// Mitsubishi GX Works2 project: Prog1 IHM_elipse_clp   PLC: FX3U/FX3UC
// Configuração Modbus RTU

PROGRAM MAIN
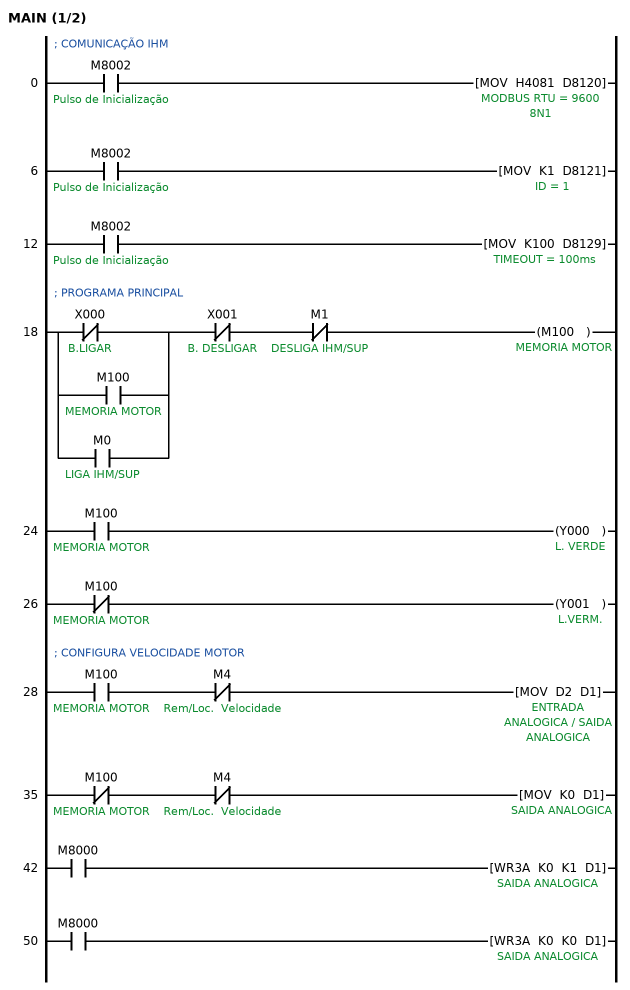
; COMUNICAÇÃO IHM
0     LD      M8002  ; Pulso de Inicialização
      MOV     H4081 D8120  ; MODBUS RTU = 9600 8N1
6     LD      M8002  ; Pulso de Inicialização
      MOV     K1 D8121  ; ID = 1
12    LD      M8002  ; Pulso de Inicialização
      MOV     K100 D8129  ; TIMEOUT = 100ms
; PROGRAMA PRINCIPAL
18    LDI     X000  ; B.LIGAR
      OR      M100  ; MEMORIA MOTOR
      OR      M0  ; LIGA IHM/SUP
      ANI     X001  ; B. DESLIGAR
      ANI     M1  ; DESLIGA IHM/SUP
      OUT     M100  ; MEMORIA MOTOR
24    LD      M100  ; MEMORIA MOTOR
      OUT     Y000  ; L. VERDE
26    LDI     M100  ; MEMORIA MOTOR
      OUT     Y001  ; L.VERM.
; CONFIGURA VELOCIDADE MOTOR
28    LD      M100  ; MEMORIA MOTOR
      ANI     M4  ; Rem/Loc.  Velocidade
      MOV     D2 D1  ; ENTRADA ANALOGICA / SAIDA ANALOGICA
35    LDI     M100  ; MEMORIA MOTOR
      ANI     M4  ; Rem/Loc.  Velocidade
      MOV     K0 D1
42    LD      M8000
      WR3A    K0 K1 D1
50    LD      M8000
      WR3A    K0 K0 D1
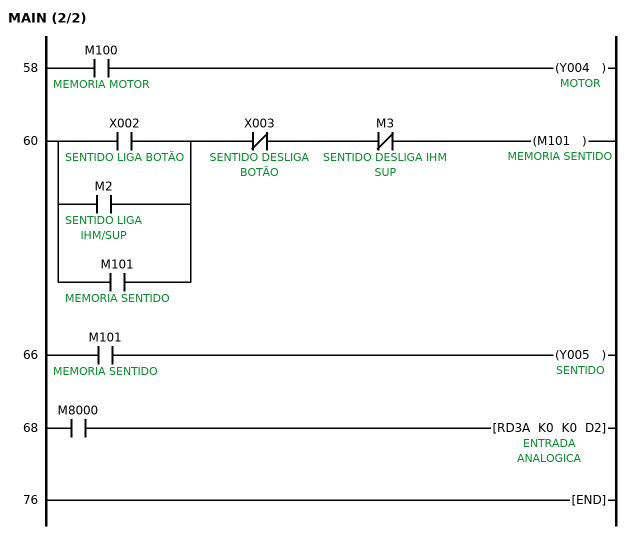
58    LD      M100  ; MEMORIA MOTOR
      OUT     Y004  ; MOTOR
60    LD      X002  ; SENTIDO LIGA BOTÃO
      OR      M2  ; SENTIDO LIGA IHM/SUP
      OR      M101  ; MEMORIA SENTIDO
      ANI     X003  ; SENTIDO DESLIGA BOTÃO
      ANI     M3  ; SENTIDO DESLIGA IHM SUP
      OUT     M101  ; MEMORIA SENTIDO
66    LD      M101  ; MEMORIA SENTIDO
      OUT     Y005  ; SENTIDO
68    LD      M8000
      RD3A    K0 K0 D2
76    END
END_PROGRAM

// device comments not shown above
Y002  ; RELE 2
M102  ; HAB. POT/SUPERV.
D0  ; REGISTRO 0
